// TIA Portal V20 export
DATA_BLOCK "PN_DEV_DIAG_PD_DB"   // DB100
{ S7_Optimized_Access := 'TRUE' }
// stored: AutoNumber false, MemoryReserve 100
   VAR
      DEVICE_DATA : "PN_DEV_DIAG_STRUCT_UDT";
   END_VAR
BEGIN
END_DATA_BLOCK
